FUNCTION TryConvert_BOOL_TO_INT : BOOL
VAR_INPUT
	in : BOOL;
	out : REFERENCE TO INT;
END_VAR

out := BOOL_TO_INT(in);
TryConvert_BOOL_TO_INT := TRUE;

END_FUNCTION

(* stored: Version 1.1.0.1, ProductVersion 3.1.4024.12
   POU TryConvert_BOOL_TO_INT: Id {9c1477e2-eaf1-4112-bc7b-42d89534a17b}, SpecialFunc None *)
